# EPICS substitutions: apps/clasTreeApp/Db/clas12Nodes.substitutions
# WARNING: DO NOT EDIT. This file was geneated at Tue Dec 15 07:08:02 EST 2015 by the a command like this:
# ./parseEpicsRecordDump [options] ioc1.dump ioc2.dump ....
# See the CLAS12 Slow Controls wiki for manuals, or the README in this directory
#
file "db/nodegraph.db" {
               pattern { P,			NPT,	TYPE }
}
